(* CoDeSys 2.3.9.55 project: ascensore.pro *)
(* Libraries: Iecsfc.lib 2.6.14 11:37:46, Standard.LIB 2.6.14 11:37:46 *)

(* Task configuration *)
TASK main (PRIORITY := 1);
	PLC_PRG();
	man();
	man_helper();
END_TASK

(* Global variable list: Global_Variables *)
VAR_GLOBAL
	(* variabili di stato*)
	stato: status;
	Start AT %IX0.0 : BOOL;
	Fine: BOOL;

	piano: ARRAY[0..2] OF floor;

	(* nell'ascensore sono comprese anche le porte*)
	elevator: ascensore;

	(* controllo manuale *)
	Mcontrol: manual;

	(* persone *)
	people: ARRAY[1..9] OF person;

END_VAR

(* Data type *)
TYPE ascensore :
STRUCT
	piano: DINT;
	occupied: BOOL;
	doorOpen: BOOL;
	doorClose: BOOL;
	FTDoor: BOOL;
	allarme:BOOL;
	allarme_col: DWORD;
	ordinata: DINT;
	doors: ARRAY[1..2] OF door;
	Masc_su: BOOL;
	Masc_giu: BOOL;
	Pin0 : BOOL;
	Pin0_col: DWORD;
	Pin1: BOOL;
	Pin1_col: DWORD;
	Pin2: BOOL;
	Pin2_col: DWORD;
END_STRUCT
END_TYPE

(* Data type *)
TYPE door :
STRUCT
	open: BOOL;
	close: BOOL;
	x_dx: DINT;
	x_sx: DINT;
	y: DINT;
	(* fotocellule *)
	porta_ft_sx1: fotocellula;
	porta_ft_dx2: fotocellula;
	porta_ft_sx2: fotocellula;
	porta_ft_dx1: fotocellula;
END_STRUCT
END_TYPE

(* Data type *)
TYPE floor :
STRUCT
	light: BOOL;
	lightcolor: DWORD;
	call: BOOL;
	callcolor: DWORD;
	ft: fotocellula;
	ftcolor: DWORD;
END_STRUCT
END_TYPE

(* Data type *)
TYPE fotocellula :
STRUCT
	status: BOOL;
	x: DINT;
	y: DINT;
END_STRUCT
END_TYPE

(* Data type *)
TYPE manual :
STRUCT
(*-Pulsanti locale tecnico-*)
	SelAM: BOOL;
	Pup: BOOL;
	Pdown: BOOL;
	Popen: BOOL;
	Pclose: BOOL;
	Res_em: BOOL;
END_STRUCT
END_TYPE

(* Data type *)
TYPE person :
STRUCT
	floor: DINT;
	status: DINT;
END_STRUCT
END_TYPE

(* Data type *)
TYPE status :
STRUCT
	off: BOOL;
	ready: BOOL;
	occupied: BOOL;
	alarm: BOOL;
	manual: BOOL;
	reset: BOOL;
END_STRUCT
END_TYPE

(* POU PLC_PRG, SFC *)
PROGRAM PLC_PRG
VAR
END_VAR
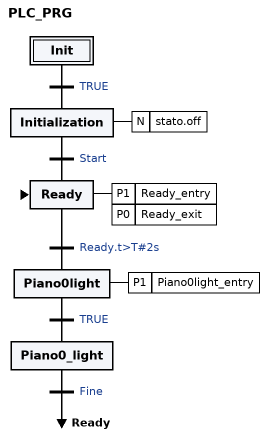
INITIAL_STEP Init:
END_STEP
TRANSITION FROM Init TO Initialization := TRUE;
END_TRANSITION
STEP Initialization:
	stato.off(N);
END_STEP
TRANSITION FROM Initialization TO Ready := Start;
END_TRANSITION
STEP Ready:
	Ready_entry(P1);
	Ready_exit(P0);
END_STEP
TRANSITION FROM Ready TO Piano0light := Ready.t>T#2s;
END_TRANSITION
STEP Piano0light:
	Piano0light_entry(P1);
END_STEP
TRANSITION FROM Piano0light TO Piano0_light := TRUE;
END_TRANSITION
STEP Piano0_light:
END_STEP
TRANSITION FROM Piano0_light TO Ready := Fine;
END_TRANSITION

ACTION Ready_entry:
(* Passaggio di inizializzazione *)

(* variabili di stato *)
stato.ready := TRUE;
stato.occupied := TRUE;
stato.alarm := TRUE;
stato.manual := TRUE;

(* controllo variabili dei piani *)
piano[0].lightcolor := 16#0000FF;
piano[0].callcolor := 16#0000FF;
piano[0].ftcolor := 16#0000FF;
piano[1].lightcolor := 16#0000FF;
piano[1].callcolor := 16#0000FF;
piano[1].ftcolor := 16#0000FF;
piano[2].lightcolor := 16#0000FF;
piano[2].callcolor := 16#0000FF;
piano[2].ftcolor := 16#0000FF;

(* controllo variabili ascensore *)
elevator.allarme_col := 16#0000FF;
elevator.Pin0_col := 16#0000FF;
elevator.Pin1_col := 16#0000FF;
elevator.Pin1_col := 16#0000FF;

(* Variabili locale tecnico *)
Mcontrol.Pup := TRUE;
Mcontrol.Pdown := TRUE;
Mcontrol.Popen := TRUE;
Mcontrol.Pclose := TRUE;
Mcontrol.Res_em := TRUE;
Mcontrol.SelAm := TRUE;
END_ACTION

ACTION Ready_exit:
(* variabili di stato *)
stato.occupied := FALSE;
stato.alarm := FALSE;
stato.manual := FALSE;

(* variabili di piano *)
piano[0].lightcolor := 16#808080;
piano[0].callcolor := 16#808080;
piano[0].ftcolor := 16#808080;
piano[1].lightcolor := 16#808080;
piano[1].callcolor := 16#808080;
piano[1].ftcolor := 16#808080;
piano[2].lightcolor := 16#808080;
piano[2].callcolor := 16#808080;
piano[2].ftcolor := 16#808080;

(* variabili ascensore *)
elevator.allarme_col := 16#808080;
elevator.Pin0_col := 16#808080;
elevator.Pin1_col := 16#808080;
elevator.Pin1_col := 16#808080;

(* Variabili locale tecnico *)
Mcontrol.Pup := FALSE;
Mcontrol.Pdown := FALSE;
Mcontrol.Popen := FALSE;
Mcontrol.Pclose := FALSE;
Mcontrol.Res_em := FALSE;
Mcontrol.SelAm := FALSE;
END_ACTION

ACTION Piano0light_entry:
piano[0].light := TRUE;
piano[0].callcolor := 16#00FF00;
piano[0].lightcolor := 16#00FF00;
piano[1].callcolor := 16#00FF00;
piano[2].callcolor := 16#00FF00;
END_ACTION
END_PROGRAM

(* POU man, LD *)
PROGRAM man
VAR
END_VAR
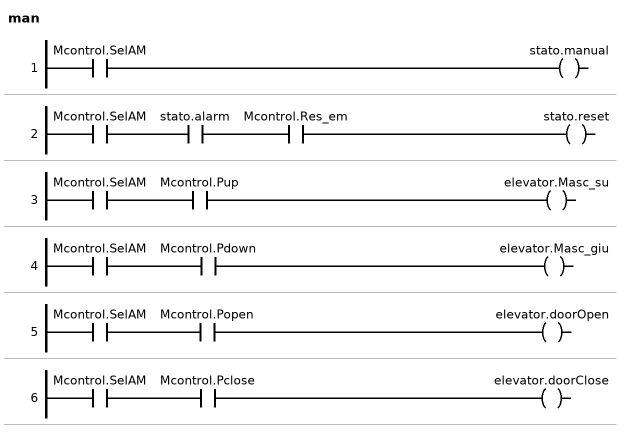
_LD_ (* Ladder Diagram *)
NETWORK 1
	[Mcontrol.SelAM] --- (stato.manual)
NETWORK 2
	[Mcontrol.SelAM] - [stato.alarm] - [Mcontrol.Res_em] --- (stato.reset)
NETWORK 3
	[Mcontrol.SelAM] - [Mcontrol.Pup] --- (elevator.Masc_su)
NETWORK 4
	[Mcontrol.SelAM] - [Mcontrol.Pdown] --- (elevator.Masc_giu)
NETWORK 5
	[Mcontrol.SelAM] - [Mcontrol.Popen] --- (elevator.doorOpen)
NETWORK 6
	[Mcontrol.SelAM] - [Mcontrol.Pclose] --- (elevator.doorClose)
_END_LD_
(* the same logic as Structured Text *)
(* Network 1 *)
stato.manual := Mcontrol.SelAM;
(* Network 2 *)
stato.reset := Mcontrol.SelAM AND stato.alarm AND Mcontrol.Res_em;
(* Network 3 *)
elevator.Masc_su := Mcontrol.SelAM AND Mcontrol.Pup;
(* Network 4 *)
elevator.Masc_giu := Mcontrol.SelAM AND Mcontrol.Pdown;
(* Network 5 *)
elevator.doorOpen := Mcontrol.SelAM AND Mcontrol.Popen;
(* Network 6 *)
elevator.doorClose := Mcontrol.SelAM AND Mcontrol.Pclose;
END_PROGRAM

(* POU man_helper, ST *)
PROGRAM man_helper
VAR
	i: DINT := 0;
END_VAR
(* Vado su di un piano *)
IF (elevator.Masc_su = TRUE) THEN
	IF (elevator.ordinata < 330) AND (i < 170) THEN
		elevator.ordinata := elevator.ordinata + 2;
		i := i + 2;
	ELSE
		i := 0;
		Mcontrol.Pup := FALSE;
	END_IF
END_IF

(* Vado giu di un piano *)
IF (elevator.Masc_giu = TRUE) THEN
	IF (elevator.ordinata > 0)  AND (i < 170) THEN
		elevator.ordinata := elevator.ordinata - 2;
		i := i + 2;
	ELSE
		i := 0;
		Mcontrol.Pdown := FALSE;
	END_IF
END_IF

(* Apro porte *)
IF (elevator.doorOpen = TRUE) THEN
	IF (elevator.doors[1].x_dx < 100) AND (elevator.doors[2].x_sx < 100) THEN
		elevator.doors[1].x_dx := elevator.doors[1].x_dx + 2;
		elevator.doors[2].x_sx := elevator.doors[2].x_sx + 2;
	ELSE
		Mcontrol.Popen := FALSE;
	END_IF
END_IF

IF (elevator.doorClose = TRUE) THEN
	IF (elevator.doors[1].x_dx > 0) AND (elevator.doors[2].x_sx > 0) THEN
		elevator.doors[1].x_dx := elevator.doors[1].x_dx - 2;
		elevator.doors[2].x_sx := elevator.doors[2].x_sx - 2;
	ELSE
		Mcontrol.Pclose := FALSE;
	END_IF
END_IF
END_PROGRAM

(* Visualisation elevator
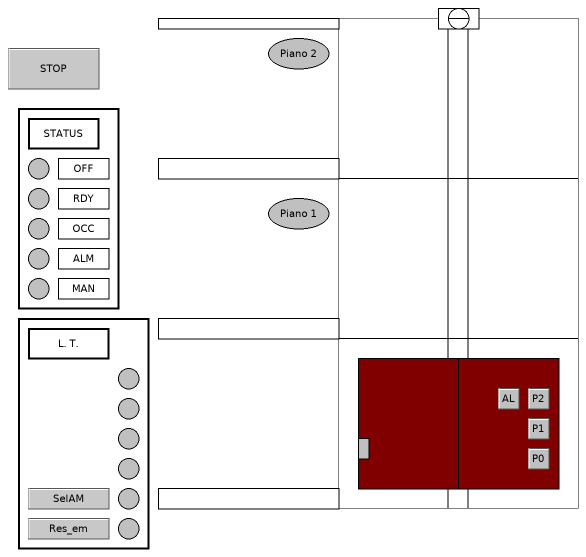
rectangle at (360,370)-(561,501): y offset -elevator.ordinata
ellipse at (270,50)-(331,81): text "Piano 2"; alarm colour if .piano2
button at (30,500)-(111,521): text "SelAM"; toggles .Mcontrol.SelAM
button at (30,530)-(111,551): text "Res_em"; toggles .Mcontrol.Res_em
ellipse at (270,210)-(331,241): text "Piano 1"; alarm colour if .piano1
rectangle at (360,370)-(461,501): right -elevator.doors[1].x_dx; y offset -elevator.ordinata
rectangle at (460,370)-(561,501): left elevator.doors[2].x_sx; y offset -elevator.ordinata
button at (530,460)-(551,481): text "P0"
button at (500,400)-(521,421): text "AL"
button at (530,430)-(551,451): text "P1"
button at (530,400)-(551,421): text "P2"
rectangle at (360,450)-(371,471): y offset -elevator.ordinata
curve at (450,30)-(470,30): angle elevator.ordinata
ellipse at (30,170)-(51,191): alarm colour if .stato.off; tooltip OFF
ellipse at (30,200)-(51,221): alarm colour if .stato.ready; tooltip READY
ellipse at (30,230)-(51,251): alarm colour if .stato.occupied; tooltip OCCUPIED
ellipse at (30,260)-(51,281): alarm colour if .stato.alarm; tooltip ALARM
ellipse at (30,290)-(51,311): alarm colour if .stato.manual; tooltip MANUAL
rectangle at (30,340)-(111,371): text "L. T."
rectangle at (60,170)-(111,191): text "OFF"
rectangle at (60,200)-(111,221): text "RDY"
rectangle at (60,230)-(111,251): text "OCC"
rectangle at (60,260)-(111,281): text "ALM"
rectangle at (60,290)-(111,311): text "MAN"
ellipse at (120,380)-(141,401): alarm colour if .Mcontrol.Pup; tooltip Pup
ellipse at (120,410)-(141,431): alarm colour if .Mcontrol.Pdown; tooltip ALARM
ellipse at (120,440)-(141,461): alarm colour if .Mcontrol.Popen; tooltip ALARM
ellipse at (120,470)-(141,491): alarm colour if .Mcontrol.Pclose; tooltip ALARM
ellipse at (120,500)-(141,521): alarm colour if .Mcontrol.SelAM; tooltip ALARM
ellipse at (120,530)-(141,551): alarm colour if .Mcontrol.Res_em; tooltip ALARM
button at (10,60)-(101,101): text "STOP"
rectangle at (30,130)-(101,161): text "STATUS"
13 more shapes without text or variables
12 elements of other kinds (tables, trends, ...) not read
*)
